// TIA Portal project "Project2" (V15)

(* hardware
DEVICE "S71500/ET200MP station_1"  S7-1500 station
   slot 0: "Rail_0"  Rack  6ES7 590-1***0-0AA0
   slot 1: "PLC_1"  CPU 1513-1 PN  6ES7 513-1AL02-0AB0  V2.5
      slot 3: "CPU display_1"  6ES7591-1AA00-0AA0
   slot 2: "DI 16x24VDC BA_1"  DI 16x24VDC BA  6ES7 521-1BH10-0AA0  V1.0
*)

// ===== PLC "PLC_1"  CPU 1513-1 PN =====

VAR_GLOBAL   // PLC tag table "Default tag table"
   "startButton" AT %I0.0 : Bool;
   "stopButton_NC" AT %I0.1 : Bool;
   "sensor1_NC" AT %I0.2 : Bool;
   "stackLight_Red" AT %Q0.0 : Bool;
   "stackLight_Green" AT %Q0.1 : Bool;
   "stackLight_Yellow" AT %Q0.2 : Bool;
   "full_level" AT %Q0.3 : Bool;
   "conv" AT %Q0.4 : Bool;
   "Clock_Byte" AT %MB0 : Byte;
   "Clock_10Hz" AT %M0.0 : Bool;
   "Clock_5Hz" AT %M0.1 : Bool;
   "Clock_2.5Hz" AT %M0.2 : Bool;
   "Clock_2Hz" AT %M0.3 : Bool;
   "Clock_1.25Hz" AT %M0.4 : Bool;
   "Clock_1Hz" AT %M0.5 : Bool;
   "Clock_0.625Hz" AT %M0.6 : Bool;
   "Clock_0.5Hz" AT %M0.7 : Bool;
   "resetButton" AT %I0.3 : Bool;
   "eStopButton_NC" AT %I0.4 : Bool;
   "sensor2_NC" AT %I0.5 : Bool;
   "conv2" AT %Q0.5 : Bool;
   "startButton_2" AT %I0.6 : Bool;
   "stopButton_NC_2" AT %I0.7 : Bool;
   "eStopButton_NC_2" AT %I1.0 : Bool;
   "resetButton_NC_2" AT %I1.1 : Bool;
   "stackLight_Red_2" AT %Q0.6 : Bool;
   "stackLight_Green_2" AT %Q0.7 : Bool;
   "stackLight_Yellow_2" AT %Q1.0 : Bool;
   "full_level_2" AT %Q1.1 : Bool;
END_VAR

TYPE "status"
   STRUCT
      running : Bool;
      full : Bool;
      ready : Bool;
      "step" : Int;
   END_STRUCT;
END_TYPE

TYPE "command"
   STRUCT
      startReq : Bool;
      resetReq : Bool;
      enable : Bool;
   END_STRUCT;
END_TYPE

TYPE "data"
   STRUCT
      count : Int;
      target : Int;
   END_STRUCT;
END_TYPE

TYPE "fault"
   STRUCT
      active : Bool;
      code : Int;
   END_STRUCT;
END_TYPE

TYPE "station"
   STRUCT
      data : "data";
      cmd : "command";
      fault : "fault";
      status : "status";
   END_STRUCT;
END_TYPE

DATA_BLOCK "PartCounter_DB"   // DB1
{ S7_Optimized_Access := 'TRUE' }
VERSION : 0.1
// stored: InstanceOfName PartCounter
"PartCounter"
BEGIN
END_DATA_BLOCK

DATA_BLOCK "StationData_DB"   // DB2
{ S7_Optimized_Access := 'TRUE' }
VERSION : 0.1
   VAR RETAIN
      station1 : "station";
      station2 : "station";
   END_VAR
BEGIN
   station1.data.target := 5;
   station2.data.target := 5;
   station1.cmd.enable := True;
END_DATA_BLOCK

DATA_BLOCK "PartCounter_DB_2"   // DB3
{ S7_Optimized_Access := 'TRUE' }
VERSION : 0.1
// stored: InstanceOfName PartCounter
"PartCounter"
BEGIN
END_DATA_BLOCK

FUNCTION_BLOCK "PartCounter"   // FB1, SCL
{ S7_Optimized_Access := 'TRUE' }
VERSION : 0.1
   VAR_INPUT
      sensor : Bool;
      stop : Bool;
      start : Bool;
      reset : Bool;
      eStopOk : Bool;
   END_VAR
   VAR_OUTPUT
      convOut : Bool;
      redLamp : Bool;
      greenLamp : Bool;
      yellowLamp : Bool;
      levelLamp : Bool;
   END_VAR
   VAR_IN_OUT
      st : "station";
   END_VAR
   VAR RETAIN
      part_counter : CTU_INT;
      timer1 : TON_TIME;
   END_VAR
   VAR
      timerStep : Bool;
      startEdge : R_TRIG;
      stopEdge : R_TRIG;
      resetEdge : R_TRIG;
   END_VAR
   VAR_TEMP
      partDetected : Bool;
      startPressed : Bool;
      stopPressed : Bool;
      counterResetPressed : Bool;
   END_VAR
BEGIN
   (*
      STATE MACHINE
      0    IDLE      — start bekle
      20   RUNNING   — konveyör çalışıyor, parça sayıyor
      30   SETTLE    — 1 sn bekleme (son parça yerleşsin)
      40   FULL      — reset bekle
      404  STOPPED   — acil çıkış, sayaç sıfırla, IDLE'a dön
   *)

   IF NOT #eStopOk THEN
       #st.status.running := FALSE;
       #st.status.step := 990;
   END_IF;
   IF #stopEdge.Q THEN
       #st.status.running := FALSE;
       #st.status.step  := 0;
   END_IF;


   // IO Normal
   #partDetected := NOT #sensor;
   #startPressed := #start;
   #stopPressed := NOT #stop;
   #counterResetPressed := #reset;


   //counter and timer def
   #part_counter(CU:= #partDetected, R:=#resetEdge.Q, PV:=#st.data.target);
   #timer1(IN := #timerStep,PT := T#1000ms);
   #startEdge(CLK := #startPressed);
   #stopEdge(CLK := #stopPressed);
   #resetEdge(CLK := #counterResetPressed);

   #st.data.count := #part_counter.CV;


   // main flow
   CASE  #st.status.step  OF


       0:
           IF (#startEdge.Q AND #st.cmd.enable) THEN
               #st.status.running := TRUE;
               #st.status.step  := 20;
           END_IF;

       20:
           IF #part_counter.QU THEN
               #timerStep := 1;
               IF #timer1.Q THEN
                   #st.status.running := FALSE;
                   #st.status.step  := 30;
               END_IF;
           END_IF;


       30:

           RESET_TIMER(#timer1);
           #timerStep := 0;
           #st.status.step  := 40;

       40:
           IF #resetEdge.Q THEN
               #st.status.step  := 0;
           END_IF;

       990: //eStop Step
           IF #eStopOk AND #resetEdge.Q THEN
               #st.status.step  := 0;
           END_IF;

           ;

       ELSE
           #st.status.step  := 0;
           ;
   END_CASE;

   // out states 
   #convOut := (#st.status.running);
   #greenLamp := ( #st.status.step =20);
   #yellowLamp := ( #st.status.step  = 40);
   #levelLamp := ( #st.status.step  = 40);
   #redLamp := ( #st.status.step  = 990);

   #st.status.full := (#st.status.step = 40);
END_FUNCTION_BLOCK

FUNCTION "factoryIO_com" : Void   // FC1, SCL
{ S7_Optimized_Access := 'TRUE' }
VERSION : 0.1
   VAR_TEMP
      I : Int;
      Value_01_DW : DWord;
      Value_02_DW : DWord;
      value : Byte;
   END_VAR
   VAR CONSTANT
      START_BYTE_IN : Int := 0;
      BYTE_COUNT_IN : Int := 63;
      START_BYTE_OUT : Int := 0;
      BYTE_COUNT_OUT : Int := 63;
      WATCHDOG_BYTE : Int := 511;
      ANALOG_OFFSET : Int := 1016;
   END_VAR
BEGIN
   // ============================================================
   // FACTORY IO DİNAMİK HABERLEŞME SÜRÜCÜSÜ
   // ============================================================

   // --- AYARLAR (Buradaki sayıları projene göre değiştir) ---
   (*
   #START_BYTE_IN := 0;   // Factory IO'da girişlerin (Inputs) başladığı byte
   #BYTE_COUNT_IN := 63;  // Kaç byte giriş okunacak? (Örn: 0 to 63)

   #START_BYTE_OUT := 0;   // Factory IO'da çıkışların (Outputs) başladığı byte
   #BYTE_COUNT_OUT := 63;  // Kaç byte çıkış yazılacak?

   #WATCHDOG_BYTE := 511; // Bağlantı kontrolü (Heartbeat) için kullanılan byte adresi
   #ANALOG_OFFSET := 1016; // Analog/DWord verilerin başladığı başlangıç adresi
   *)

   // --------------------------------------------------------

   REGION 1_WATCHDOG
       // Bağlantının koptuğunu anlamak için Q adresindeki sayaç
       #value := PEEK(area := 16#82, dbNumber := 0, byteOffset := #WATCHDOG_BYTE);
       #value := #value + 1;
       POKE(area := 16#82,
            dbNumber := 0,
            byteOffset := #WATCHDOG_BYTE,
            value := #value);
   END_REGION

   REGION 2_INPUT_SYNC
       // Girişleri Factory IO'dan PLC'ye aktarır
       FOR #I := 0 TO #BYTE_COUNT_IN DO
           // Kaynaktan oku (Genellikle 16#81: Inputs)
           #value := PEEK(area := 16#81, dbNumber := 0, byteOffset := #START_BYTE_IN + #I);

           // Hedefe yaz (16#1: Process Image Input)
           POKE(area := 16#1,
                dbNumber := 0,
                byteOffset := #START_BYTE_IN + #I,
                value := #value);
       END_FOR;
   END_REGION

   REGION 3_ANALOG_DATA
       // DWord veya Analog verileri yazar (DW#1 ve DW#2)
       POKE(area := 16#82,
            dbNumber := 0,
            byteOffset := #ANALOG_OFFSET,
            value := #Value_01_DW);
       POKE(area := 16#82,
            dbNumber := 0,
            byteOffset := #ANALOG_OFFSET + 4,
            value := #Value_02_DW);
   END_REGION
END_FUNCTION

ORGANIZATION_BLOCK "Main"   // OB1, SCL, ProgramCycle
TITLE = "Main Program Sweep (Cycle)"
{ S7_Optimized_Access := 'TRUE' }
VERSION : 0.1
   VAR_INPUT
      Initial_Call : Bool;   // Initial call of this OB
      Remanence : Bool;   // =True, if remanent data are available
   END_VAR
BEGIN
   REGION Factory_IO
       // Get inputs from factory io 

       "factoryIO_com"();

   END_REGION



   "PartCounter_DB"(sensor := "sensor1_NC",
                    stop := "stopButton_NC",
                    start := "startButton",
                    reset := "resetButton",
                    eStopOk := "eStopButton_NC",
                    st:= "StationData_DB".station1,
                    convOut => "conv",
                    redLamp => "stackLight_Red",
                    greenLamp => "stackLight_Green",
                    yellowLamp => "stackLight_Yellow",
                    levelLamp => "full_level");

   "PartCounter_DB_2"(sensor:="sensor2_NC",
                      stop:="stopButton_NC_2",
                      start:="startButton_2",
                      reset:="resetButton_NC_2",
                      eStopOk:="eStopButton_NC",
                      convOut=>"conv2",
                      redLamp=>"stackLight_Red_2",
                      greenLamp=>"stackLight_Green_2",
                      yellowLamp=>"stackLight_Yellow_2",
                      levelLamp=>"full_level_2",
                      st:="StationData_DB".station2);

   "StationData_DB".station2.cmd.enable := "StationData_DB".station1.status.full;
END_ORGANIZATION_BLOCK